FUNCTION_BLOCK FB_CalcFocalLengthLensSetMock EXTENDS FB_FalliblePublicMock IMPLEMENTS I_CalcFocalLengthLensSet
VAR
    fbFocalLength : FB_QuantityLREALPublic(Units := 'm');
END_VAR


METHOD Calculate
VAR_INPUT
    LensSet : I_LensSet;
END_VAR
VAR_IN_OUT
    FocalLength : FB_QuantityLREALPublic(Units := 'm');
END_VAR

FocalLength := fbFocalLength;
END_METHOD


METHOD SetResult
VAR_INPUT
    Result : I_QuantityLREAL;
END_VAR

fbFocalLength.Copy(QuantityToCopy := Result);
END_METHOD


METHOD SetValid

fbFocalLength.Val := 1.0;
fbFocalLength.Units := 'm';
fbFocalLength.ClearError();
ClearError();
END_METHOD

END_FUNCTION_BLOCK

(* stored: Version 1.1.0.1
   POU FB_CalcFocalLengthLensSetMock: Id {db9e08db-5cbf-4afa-b31b-28bcb5b02fc5}, SpecialFunc None
   Method Calculate: Id {9449408e-a2a8-4a84-848f-08f055b3b183}
   Method SetResult: Id {b90caf58-8ba2-4f62-ae29-0aec1937810d}
   Method SetValid: Id {4f9c11d6-93e5-42e8-a4e7-e7a7d4a383f5} *)
